	LOCAL CONST Robtarget Tr_meulage_bavure_P251 :=[[98.1400390625,117.987203125,73.8456328125],[0.127040389675562,-0.107005563499621,0.63527191816149,-0.754214915502625],[0,0,0,0],[8.999999E+09,8.999999E+09,8.999999E+09,8.999999E+09,8.999999E+09,8.999999E+09]];
	LOCAL CONST Robtarget Tr_meulage_bavure_P252 :=[[98.0491484375,117.9515,73.860046875],[0.172195881687435,-0.145894069896958,0.629753687846079,-0.74328580730635],[0,0,0,0],[8.999999E+09,8.999999E+09,8.999999E+09,8.999999E+09,8.999999E+09,8.999999E+09]];
	LOCAL CONST Robtarget Tr_meulage_bavure_P253 :=[[95.44875,117.0130703125,74.2617890625],[0.207950204557917,-0.177032849806687,0.623590925198428,-0.73249603447651],[0,0,0,0],[8.999999E+09,8.999999E+09,8.999999E+09,8.999999E+09,8.999999E+09,8.999999E+09]];
	LOCAL CONST Robtarget Tr_meulage_bavure_P254 :=[[94.7231171875,116.4957578125,74.4063515625],[0.235260133644742,-0.200979067526871,0.617662145956152,-0.72301698277864],[0,0,0,0],[8.999999E+09,8.999999E+09,8.999999E+09,8.999999E+09,8.999999E+09,8.999999E+09]];
	LOCAL CONST Robtarget Tr_meulage_bavure_P255 :=[[94.14340625,116.1705234375,74.51065625],[0.255147496976429,-0.218409662757732,0.612521728241192,-0.715551609901858],[0,0,0,0],[8.999999E+09,8.999999E+09,8.999999E+09,8.999999E+09,8.999999E+09,8.999999E+09]];
	LOCAL CONST Robtarget Tr_meulage_bavure_P256 :=[[93.2889140625,115.3411484375,74.708875],[0.268575710211451,-0.230015700629152,0.608452712166897,-0.710454194445527],[0,0,0,0],[8.999999E+09,8.999999E+09,8.999999E+09,8.999999E+09,8.999999E+09,8.999999E+09]];
	LOCAL CONST Robtarget Tr_meulage_bavure_P257 :=[[90.7856171875,112.887015625,75.292671875],[0.276376961310427,-0.236441862806716,0.605550122499022,-0.707827712025126],[0,0,0,0],[8.999999E+09,8.999999E+09,8.999999E+09,8.999999E+09,8.999999E+09,8.999999E+09]];
	LOCAL CONST Robtarget Tr_meulage_bavure_P258 :=[[88.863078125,110.5822109375,75.79440625],[0.279245959102819,-0.238275525006702,0.603780767368518,-0.707598228844173],[0,0,0,0],[8.999999E+09,8.999999E+09,8.999999E+09,8.999999E+09,8.999999E+09,8.999999E+09]];
	LOCAL CONST Robtarget Tr_meulage_bavure_P259 :=[[86.18025,107.824984375,76.4362265625],[0.277632487950623,-0.235945820214436,0.603068641778131,-0.709618196540621],[0,0,0,0],[8.999999E+09,8.999999E+09,8.999999E+09,8.999999E+09,8.999999E+09,8.999999E+09]];
	LOCAL CONST Robtarget Tr_meulage_bavure_P260 :=[[80.36984375,101.8534296875,77.8262578125],[0.27163574756326,-0.229638288909727,0.603381148543333,-0.713730668035842],[0,0,0,0],[8.999999E+09,8.999999E+09,8.999999E+09,8.999999E+09,8.999999E+09,8.999999E+09]];
	LOCAL CONST Robtarget Tr_meulage_bavure_P261 :=[[77.1337109375,98.5814375,78.59359375],[0.260925476383616,-0.219208728105446,0.60474203438692,-0.719828105273714],[0,0,0,0],[8.999999E+09,8.999999E+09,8.999999E+09,8.999999E+09,8.999999E+09,8.999999E+09]];
	LOCAL CONST Robtarget Tr_meulage_bavure_P262 :=[[72.1760859375,93.4272109375,79.787125],[0.244696261183989,-0.204145790459714,0.607216023498567,-0.727830293960579],[0,0,0,0],[8.999999E+09,8.999999E+09,8.999999E+09,8.999999E+09,8.999999E+09,8.999999E+09]];
	LOCAL CONST Robtarget Tr_meulage_bavure_P263 :=[[71.50584375,92.7481328125,79.946234375],[0.221726143472033,-0.183626372472933,0.610829559169254,-0.737567706911403],[0,0,0,0],[8.999999E+09,8.999999E+09,8.999999E+09,8.999999E+09,8.999999E+09,8.999999E+09]];
	LOCAL CONST Robtarget Tr_meulage_bavure_P264 :=[[71.2399140625,92.5131875,80.0049765625],[0.190628848170377,-0.156707517312216,0.615389383499725,-0.748598225311084],[0,0,0,0],[8.999999E+09,8.999999E+09,8.999999E+09,8.999999E+09,8.999999E+09,8.999999E+09]];
	LOCAL CONST Robtarget Tr_meulage_bavure_P265 :=[[70.7853359375,92.1913046875,80.0952578125],[0.150575822021713,-0.122909725316936,0.620287722757024,-0.759910035623892],[0,0,0,0],[8.999999E+09,8.999999E+09,8.999999E+09,8.999999E+09,8.999999E+09,8.999999E+09]];
	LOCAL CONST Robtarget Tr_meulage_bavure_P266 :=[[68.07696875,90.16765625,80.6466328125],[0.102447611715575,-0.0830907118710058,0.624412481473696,-0.769876271510173],[0,0,0,0],[8.999999E+09,8.999999E+09,8.999999E+09,8.999999E+09,8.999999E+09,8.999999E+09]];
	LOCAL CONST Robtarget Tr_meulage_bavure_P267 :=[[65.683109375,88.9370859375,81.0630625],[0.0497692839972195,-0.0401467777631947,0.626564781602221,-0.776741803343555],[0,0,0,0],[8.999999E+09,8.999999E+09,8.999999E+09,8.999999E+09,8.999999E+09,8.999999E+09]];
	LOCAL CONST Robtarget Tr_meulage_bavure_P268 :=[[64.74205859375,88.55846875,81.21340625],[0.001363095089986,-0.00109499953132052,-0.626270337472808,0.779604006755672],[0,0,0,0],[8.999999E+09,8.999999E+09,8.999999E+09,8.999999E+09,8.999999E+09,8.999999E+09]];
	LOCAL CONST Robtarget Tr_meulage_bavure_P269 :=[[62.3850234375,88.1528203125,81.5210078125],[0.0437419301601574,-0.0350453753396799,-0.624275842926536,0.779190693701823],[0,0,0,0],[8.999999E+09,8.999999E+09,8.999999E+09,8.999999E+09,8.999999E+09,8.999999E+09]];
	LOCAL CONST Robtarget Tr_meulage_bavure_P270 :=[[61.54280859375,88.344234375,81.5881796875],[0.0710459531376083,-0.0568640478748205,-0.622285158362753,0.777483205145618],[0,0,0,0],[8.999999E+09,8.999999E+09,8.999999E+09,8.999999E+09,8.999999E+09,8.999999E+09]];
	LOCAL CONST Robtarget Tr_meulage_bavure_P271 :=[[59.371765625,88.1027109375,81.85471875],[0.0786620779021897,-0.0630080775834088,-0.621986088766345,0.776515012759249],[0,0,0,0],[8.999999E+09,8.999999E+09,8.999999E+09,8.999999E+09,8.999999E+09,8.999999E+09]];
	LOCAL CONST Robtarget Tr_meulage_bavure_P272 :=[[56.79593359375,90.4163515625,81.840546875],[0.064068817064071,-0.0514508699376922,-0.624029588381331,0.777068251498729],[0,0,0,0],[8.999999E+09,8.999999E+09,8.999999E+09,8.999999E+09,8.999999E+09,8.999999E+09]];
	LOCAL CONST Robtarget Tr_meulage_bavure_P273 :=[[48.6920625,97.4299765625,81.8296640625],[0.0277015568674016,-0.0223423861530457,-0.62739597405027,0.777886709793671],[0,0,0,0],[8.999999E+09,8.999999E+09,8.999999E+09,8.999999E+09,8.999999E+09,8.999999E+09]];
	LOCAL CONST Robtarget Tr_meulage_bavure_P274 :=[[47.0812421875,97.794265625,81.9583671875],[0.0252356318326453,-0.0204756378074699,0.629734896885263,-0.776130060484254],[0,0,0,0],[8.999999E+09,8.999999E+09,8.999999E+09,8.999999E+09,8.999999E+09,8.999999E+09]];
	LOCAL CONST Robtarget Tr_meulage_bavure_P275 :=[[44.806,97.7003515625,82.21746875],[0.0848193325394842,-0.0693367803526094,0.629095491043596,-0.769569330773068],[0,0,0,0],[8.999999E+09,8.999999E+09,8.999999E+09,8.999999E+09,8.999999E+09,8.999999E+09]];
	LOCAL CONST Robtarget Tr_meulage_bavure_P276 :=[[42.50455859375,97.2184921875,82.52871875],[0.140587062127015,-0.115938530664608,0.625580695787566,-0.758579150865466],[0,0,0,0],[8.999999E+09,8.999999E+09,8.999999E+09,8.999999E+09,8.999999E+09,8.999999E+09]];
	LOCAL CONST Robtarget Tr_meulage_bavure_P277 :=[[39.54287109375,95.636578125,83.0514765625],[0.186282650440504,-0.155136411224339,0.620854079163028,-0.745500959384978],[0,0,0,0],[8.999999E+09,8.999999E+09,8.999999E+09,8.999999E+09,8.999999E+09,8.999999E+09]];
	LOCAL CONST Robtarget Tr_meulage_bavure_P278 :=[[39.0804296875,95.4284609375,83.1281640625],[0.220511472840555,-0.185597052614264,0.616612847403539,-0.732609732957109],[0,0,0,0],[8.999999E+09,8.999999E+09,8.999999E+09,8.999999E+09,8.999999E+09,8.999999E+09]];
	LOCAL CONST Robtarget Tr_meulage_bavure_P279 :=[[38.82609765625,95.2573359375,83.1775390625],[0.244591306708348,-0.208162312657775,0.613779305281082,-0.721192421396913],[0,0,0,0],[8.999999E+09,8.999999E+09,8.999999E+09,8.999999E+09,8.999999E+09,8.999999E+09]];
	LOCAL CONST Robtarget Tr_meulage_bavure_P280 :=[[35.845515625,92.55171875,83.845140625],[0.260660984276943,-0.224358974738056,0.612563122723334,-0.711677822058339],[0,0,0,0],[8.999999E+09,8.999999E+09,8.999999E+09,8.999999E+09,8.999999E+09,8.999999E+09]];
	LOCAL CONST Robtarget Tr_meulage_bavure_P281 :=[[32.57470703125,88.9592421875,84.65696875],[0.270796308543816,-0.235720468748974,0.61279461348127,-0.703980100272833],[0,0,0,0],[8.999999E+09,8.999999E+09,8.999999E+09,8.999999E+09,8.999999E+09,8.999999E+09]];
	LOCAL CONST Robtarget Tr_meulage_bavure_P282 :=[[32.4998046875,88.8786796875,84.67534375],[0.276769983598911,-0.243580619288763,0.614120686336212,-0.697798424116522],[0,0,0,0],[8.999999E+09,8.999999E+09,8.999999E+09,8.999999E+09,8.999999E+09,8.999999E+09]];
	LOCAL CONST Robtarget Tr_meulage_bavure_P283 :=[[32.41517578125,88.7886328125,84.6959765625],[0.279976048156399,-0.249000355415884,0.616150254112905,-0.692799465803844],[0,0,0,0],[8.999999E+09,8.999999E+09,8.999999E+09,8.999999E+09,8.999999E+09,8.999999E+09]];
	LOCAL CONST Robtarget Tr_meulage_bavure_P284 :=[[32.27737890625,88.6504765625,84.7285078125],[0.281492307641199,-0.252818582194378,0.618524049054791,-0.688674702582376],[0,0,0,0],[8.999999E+09,8.999999E+09,8.999999E+09,8.999999E+09,8.999999E+09,8.999999E+09]];
	LOCAL CONST Robtarget Tr_meulage_bavure_P285 :=[[28.927525390625,85.261125,85.523109375],[0.282090145605153,-0.255653636684952,0.620965252888204,-0.685177730598208],[0,0,0,0],[8.999999E+09,8.999999E+09,8.999999E+09,8.999999E+09,8.999999E+09,8.999999E+09]];
	LOCAL CONST Robtarget Tr_meulage_bavure_P286 :=[[21.47466796875,77.75175,87.286984375],[0.282327813795655,-0.257956584167709,0.623251031261927,-0.682134560239282],[0,0,0,0],[8.999999E+09,8.999999E+09,8.999999E+09,8.999999E+09,8.999999E+09,8.999999E+09]];
	LOCAL CONST Robtarget Tr_meulage_bavure_P287 :=[[21.25967578125,77.5322421875,87.338234375],[0.282601819625309,-0.260063837576601,0.625225023955301,-0.679409067756303],[0,0,0,0],[8.999999E+09,8.999999E+09,8.999999E+09,8.999999E+09,8.999999E+09,8.999999E+09]];
	LOCAL CONST Robtarget Tr_meulage_bavure_P288 :=[[20.5857109375,76.868484375,87.495796875],[0.283101282414858,-0.26214225566945,0.626816081849102,-0.67693182908099],[0,0,0,0],[8.999999E+09,8.999999E+09,8.999999E+09,8.999999E+09,8.999999E+09,8.999999E+09]];
	LOCAL CONST Robtarget Tr_meulage_bavure_P289 :=[[16.90142578125,73.2369765625,88.3575],[0.283868643218972,-0.264223838178046,0.628004469387492,-0.674696037608653],[0,0,0,0],[8.999999E+09,8.999999E+09,8.999999E+09,8.999999E+09,8.999999E+09,8.999999E+09]];
	LOCAL CONST Robtarget Tr_meulage_bavure_P290 :=[[15.873087890625,72.23375,88.5966953125],[0.284822251592282,-0.26622897396762,0.628823532756499,-0.672740204737079],[0,0,0,0],[8.999999E+09,8.999999E+09,8.999999E+09,8.999999E+09,8.999999E+09,8.999999E+09]];
	LOCAL CONST Robtarget Tr_meulage_bavure_P291 :=[[15.2935966796875,71.60771875,88.739203125],[0.285799359935917,-0.268004907206124,0.629345060745857,-0.671131052841732],[0,0,0,0],[8.999999E+09,8.999999E+09,8.999999E+09,8.999999E+09,8.999999E+09,8.999999E+09]];
	LOCAL CONST Robtarget Tr_meulage_bavure_P292 :=[[12.464833984375,68.6040234375,89.4281953125],[0.286627272536143,-0.269395860937951,0.629654783981739,-0.669929496109032],[0,0,0,0],[8.999999E+09,8.999999E+09,8.999999E+09,8.999999E+09,8.999999E+09,8.999999E+09]];
	LOCAL CONST Robtarget Tr_meulage_bavure_P293 :=[[12.3877333984375,68.5313046875,89.4458046875],[0.287172673957076,-0.270282218475825,0.629822260816589,-0.669181064800857],[0,0,0,0],[8.999999E+09,8.999999E+09,8.999999E+09,8.999999E+09,8.999999E+09,8.999999E+09]];
	LOCAL CONST Robtarget Tr_meulage_bavure_P294 :=[[12.30885546875,68.4598515625,89.463453125],[0.287361487578792,-0.270586373771854,0.629876519961336,-0.668925974519527],[0,0,0,0],[8.999999E+09,8.999999E+09,8.999999E+09,8.999999E+09,8.999999E+09,8.999999E+09]];
	LOCAL CONST Robtarget Tr_meulage_bavure_degg1 :=[[5.0687653180683,75.3315448036295,88.8626814463921],[0.287361487578792,-0.270586373771854,0.629876519961336,-0.668925974519527],[0,0,0,0],[8.999999E+09,8.999999E+09,8.999999E+09,8.999999E+09,8.999999E+09,8.999999E+09]];
	LOCAL CONST Robtarget Tr_meulage_bavure_degg2 :=[[-132.492947544884,205.89371638509,77.4480195528422],[0.287361487578792,-0.270586373771854,0.629876519961336,-0.668925974519527],[0,0,0,0],[8.999999E+09,8.999999E+09,8.999999E+09,8.999999E+09,8.999999E+09,8.999999E+09]];
	LOCAL PROC Tr_pick()
		!!Programme Tr_pick - 11/05/2023 15:21:44;
		 CONST Robtarget Ppick :=[[54.302843354765,-14.0729442667339,117.853362865586],[0.0438323717266724,0.92362905790366,0.371077115821677,-0.0853806810600477],[0,0,0,0],[8.999999E+09,8.999999E+09,8.999999E+09,8.999999E+09,8.999999E+09,8.999999E+09]];
		 VAR Pose Ref :=[[0,0,0],[1,0,0,0]];
		LocalisationPieceTable 80 \model:=0;
		MoveJ Reltool(Ppick,0,0,-200),V1000,Z0,Tool_Prehenseur_1 \Wobj:=Wobj_vision;
		MoveL Reltool(Ppick,0,0,-100),V500,Z0,Tool_Prehenseur_1 \Wobj:=Wobj_vision;
		MoveL Reltool(Ppick,0,0,-10),V200,Z0,Tool_Prehenseur_1 \Wobj:=Wobj_vision;
		MoveL Ppick,V100,Fine,Tool_Prehenseur_1 \Wobj:=Wobj_vision;
		Gripper_Close;
		MoveL Reltool(Ppick,0,0,-200),V500,Z0,Tool_Prehenseur_1 \Wobj:=Wobj_vision;
		LocalisationPiecePrehenseur 80 \model:=0,Ref;
	ENDPROC
	LOCAL PROC Tr_Cut()
		!!Programme Tr_Cut - 11/05/2023 15:21:44;
		confJ \off;
		confL \off;
		Tool := ToolOffset(Tool_M2_D490_S180);
	ENDPROC
	LOCAL PROC Tr_meulage_motif_1()
		!!Programme Tr_meulage_motif_1 - 11/05/2023 15:21:44;
		 CONST Speeddata vitesse_Meulage :=[50, 500, 0, 0];
		confJ \off;
		confL \off;
		Tool := ToolOffset(Tool_M1_D500_S0);
		MoveAbsJ [[0,-40,40,0,90,0],[8.999999E+09,8.999999E+09,8.999999E+09,8.999999E+09,8.999999E+09,8.999999E+09]] ,V1000,Z0,Tool_M1_D500_S0 \Wobj:=Wobj_Part_0;
		MoveJ Tr_meulage_motif_1_App1,V2000,Z100,Tool,\Wobj:=Wobj_Part_0;
		MoveJ Tr_meulage_motif_1_App2,V500,Z0,Tool,\Wobj:=Wobj_Part_0;
		MoveL Tr_meulage_motif_1_P0,[12.5,500,0,0],z0,Tool \wobj:=Wobj_Part_0;
		MoveL Tr_meulage_motif_1_P1,[12.5,500,0,0],z0,Tool \wobj:=Wobj_Part_0;
		MoveL Tr_meulage_motif_1_P2,[12.5,500,0,0],z0,Tool \wobj:=Wobj_Part_0;
		MoveL Tr_meulage_motif_1_P3,[12.5,500,0,0],z0,Tool \wobj:=Wobj_Part_0;
		MoveL Tr_meulage_motif_1_P4,[12.5,500,0,0],z0,Tool \wobj:=Wobj_Part_0;
		MoveL Tr_meulage_motif_1_P5,[12.5,500,0,0],z0,Tool \wobj:=Wobj_Part_0;
		MoveL Tr_meulage_motif_1_P6,[12.5,500,0,0],z0,Tool \wobj:=Wobj_Part_0;
		MoveL Tr_meulage_motif_1_P7,[12.5,500,0,0],z0,Tool \wobj:=Wobj_Part_0;
		MoveL Tr_meulage_motif_1_P8,[12.5,500,0,0],z0,Tool \wobj:=Wobj_Part_0;
		MoveL Tr_meulage_motif_1_P9,[12.5,500,0,0],z0,Tool \wobj:=Wobj_Part_0;
		MoveL Tr_meulage_motif_1_P10,[12.5,500,0,0],z0,Tool \wobj:=Wobj_Part_0;
		MoveL Tr_meulage_motif_1_P11,[12.5,500,0,0],z0,Tool \wobj:=Wobj_Part_0;
		MoveL Tr_meulage_motif_1_P12,[12.5,500,0,0],z0,Tool \wobj:=Wobj_Part_0;
		MoveL Tr_meulage_motif_1_P13,[12.5,500,0,0],z0,Tool \wobj:=Wobj_Part_0;
		MoveL Tr_meulage_motif_1_P14,[12.5,500,0,0],z0,Tool \wobj:=Wobj_Part_0;
		MoveL Tr_meulage_motif_1_P15,[12.5,500,0,0],z0,Tool \wobj:=Wobj_Part_0;
		MoveL Tr_meulage_motif_1_P16,[12.5,500,0,0],z0,Tool \wobj:=Wobj_Part_0;
		MoveL Tr_meulage_motif_1_P17,[12.5,500,0,0],z0,Tool \wobj:=Wobj_Part_0;
		MoveL Tr_meulage_motif_1_P18,[12.5,500,0,0],z0,Tool \wobj:=Wobj_Part_0;
		MoveL Tr_meulage_motif_1_P19,[12.5,500,0,0],z0,Tool \wobj:=Wobj_Part_0;
		MoveL Tr_meulage_motif_1_P20,[12.5,500,0,0],z0,Tool \wobj:=Wobj_Part_0;
		MoveL Tr_meulage_motif_1_P21,[12.5,500,0,0],z0,Tool \wobj:=Wobj_Part_0;
		MoveL Tr_meulage_motif_1_P22,[12.5,500,0,0],z0,Tool \wobj:=Wobj_Part_0;
		MoveL Tr_meulage_motif_1_P23,[12.5,500,0,0],z0,Tool \wobj:=Wobj_Part_0;
		MoveL Tr_meulage_motif_1_P24,[12.5,500,0,0],z0,Tool \wobj:=Wobj_Part_0;
		MoveL Tr_meulage_motif_1_P25,[12.5,500,0,0],z0,Tool \wobj:=Wobj_Part_0;
		MoveL Tr_meulage_motif_1_P26,[12.5,500,0,0],z0,Tool \wobj:=Wobj_Part_0;
		MoveL Tr_meulage_motif_1_P27,[12.5,500,0,0],z0,Tool \wobj:=Wobj_Part_0;
		MoveL Tr_meulage_motif_1_P28,[12.5,500,0,0],z0,Tool \wobj:=Wobj_Part_0;
		MoveL Tr_meulage_motif_1_P29,[12.5,500,0,0],z0,Tool \wobj:=Wobj_Part_0;
		MoveL Tr_meulage_motif_1_P30,[12.5,500,0,0],z0,Tool \wobj:=Wobj_Part_0;
		MoveL Tr_meulage_motif_1_P31,[12.5,500,0,0],z0,Tool \wobj:=Wobj_Part_0;
		MoveL Tr_meulage_motif_1_P32,[12.5,500,0,0],z0,Tool \wobj:=Wobj_Part_0;
		MoveL Tr_meulage_motif_1_P33,[12.5,500,0,0],z0,Tool \wobj:=Wobj_Part_0;
		MoveL Tr_meulage_motif_1_P34,[12.5,500,0,0],z0,Tool \wobj:=Wobj_Part_0;
		MoveL Tr_meulage_motif_1_P35,[12.5,500,0,0],z0,Tool \wobj:=Wobj_Part_0;
		MoveL Tr_meulage_motif_1_P36,[12.5,500,0,0],z0,Tool \wobj:=Wobj_Part_0;
		MoveL Tr_meulage_motif_1_P37,[12.5,500,0,0],z0,Tool \wobj:=Wobj_Part_0;
		MoveL Tr_meulage_motif_1_P38,[12.5,500,0,0],z0,Tool \wobj:=Wobj_Part_0;
		MoveL Tr_meulage_motif_1_P39,[12.5,500,0,0],z0,Tool \wobj:=Wobj_Part_0;
		MoveL Tr_meulage_motif_1_P40,[12.5,500,0,0],z0,Tool \wobj:=Wobj_Part_0;
		MoveL Tr_meulage_motif_1_P41,[12.5,500,0,0],z0,Tool \wobj:=Wobj_Part_0;
		MoveL Tr_meulage_motif_1_P42,[12.5,500,0,0],z0,Tool \wobj:=Wobj_Part_0;
		MoveL Tr_meulage_motif_1_P43,[12.5,500,0,0],z0,Tool \wobj:=Wobj_Part_0;
		MoveL Tr_meulage_motif_1_P44,[12.5,500,0,0],z0,Tool \wobj:=Wobj_Part_0;
		MoveL Tr_meulage_motif_1_P45,[12.5,500,0,0],z0,Tool \wobj:=Wobj_Part_0;
		MoveL Tr_meulage_motif_1_P46,[12.5,500,0,0],z0,Tool \wobj:=Wobj_Part_0;
		MoveL Tr_meulage_motif_1_P47,[12.5,500,0,0],z0,Tool \wobj:=Wobj_Part_0;
		MoveL Tr_meulage_motif_1_P48,[12.5,500,0,0],z0,Tool \wobj:=Wobj_Part_0;
		MoveL Tr_meulage_motif_1_P49,[12.5,500,0,0],z0,Tool \wobj:=Wobj_Part_0;
		MoveL Tr_meulage_motif_1_P50,[12.5,500,0,0],z0,Tool \wobj:=Wobj_Part_0;
		MoveL Tr_meulage_motif_1_P51,[12.5,500,0,0],z0,Tool \wobj:=Wobj_Part_0;
		MoveL Tr_meulage_motif_1_P52,[12.5,500,0,0],z0,Tool \wobj:=Wobj_Part_0;
		MoveL Tr_meulage_motif_1_P53,[12.5,500,0,0],z0,Tool \wobj:=Wobj_Part_0;
		MoveL Tr_meulage_motif_1_P54,[12.5,500,0,0],z0,Tool \wobj:=Wobj_Part_0;
		MoveL Tr_meulage_motif_1_P55,[12.5,500,0,0],z0,Tool \wobj:=Wobj_Part_0;
		MoveL Tr_meulage_motif_1_P56,[12.5,500,0,0],z0,Tool \wobj:=Wobj_Part_0;
		MoveL Tr_meulage_motif_1_P57,[12.5,500,0,0],z0,Tool \wobj:=Wobj_Part_0;
		MoveL Tr_meulage_motif_1_P58,[12.5,500,0,0],z0,Tool \wobj:=Wobj_Part_0;
		MoveL Tr_meulage_motif_1_P59,[12.5,500,0,0],z0,Tool \wobj:=Wobj_Part_0;
		MoveL Tr_meulage_motif_1_P60,[12.5,500,0,0],z0,Tool \wobj:=Wobj_Part_0;
		MoveL Tr_meulage_motif_1_P61,[12.5,500,0,0],z0,Tool \wobj:=Wobj_Part_0;
		MoveL Tr_meulage_motif_1_P62,[12.5,500,0,0],z0,Tool \wobj:=Wobj_Part_0;
		MoveL Tr_meulage_motif_1_P63,[12.5,500,0,0],z0,Tool \wobj:=Wobj_Part_0;
		MoveL Tr_meulage_motif_1_P64,[12.5,500,0,0],z0,Tool \wobj:=Wobj_Part_0;
		MoveL Tr_meulage_motif_1_P65,[12.5,500,0,0],z0,Tool \wobj:=Wobj_Part_0;
		MoveL Tr_meulage_motif_1_P66,[12.5,500,0,0],z0,Tool \wobj:=Wobj_Part_0;
		MoveL Tr_meulage_motif_1_P67,[12.5,500,0,0],z0,Tool \wobj:=Wobj_Part_0;
		MoveL Tr_meulage_motif_1_P68,[12.5,500,0,0],z0,Tool \wobj:=Wobj_Part_0;
		MoveL Tr_meulage_motif_1_P69,[12.5,500,0,0],z0,Tool \wobj:=Wobj_Part_0;
		MoveL Tr_meulage_motif_1_P70,[12.5,500,0,0],z0,Tool \wobj:=Wobj_Part_0;
		MoveL Tr_meulage_motif_1_P71,[12.5,500,0,0],z0,Tool \wobj:=Wobj_Part_0;
		MoveL Tr_meulage_motif_1_P72,[12.5,500,0,0],z0,Tool \wobj:=Wobj_Part_0;
		MoveL Tr_meulage_motif_1_P73,[12.5,500,0,0],z0,Tool \wobj:=Wobj_Part_0;
		MoveL Tr_meulage_motif_1_P74,[12.5,500,0,0],z0,Tool \wobj:=Wobj_Part_0;
		MoveL Tr_meulage_motif_1_P75,[12.5,500,0,0],z0,Tool \wobj:=Wobj_Part_0;
		MoveL Tr_meulage_motif_1_P76,[12.5,500,0,0],z0,Tool \wobj:=Wobj_Part_0;
		MoveL Tr_meulage_motif_1_P77,[12.5,500,0,0],z0,Tool \wobj:=Wobj_Part_0;
		MoveL Tr_meulage_motif_1_P78,[12.5,500,0,0],z0,Tool \wobj:=Wobj_Part_0;
		MoveL Tr_meulage_motif_1_P79,[12.5,500,0,0],z0,Tool \wobj:=Wobj_Part_0;
		MoveL Tr_meulage_motif_1_P80,[12.5,500,0,0],z0,Tool \wobj:=Wobj_Part_0;
		MoveL Tr_meulage_motif_1_P81,[12.5,500,0,0],z0,Tool \wobj:=Wobj_Part_0;
		MoveL Tr_meulage_motif_1_P82,[12.5,500,0,0],z0,Tool \wobj:=Wobj_Part_0;
		MoveL Tr_meulage_motif_1_P83,[12.5,500,0,0],z0,Tool \wobj:=Wobj_Part_0;
		MoveL Tr_meulage_motif_1_P84,[12.5,500,0,0],z0,Tool \wobj:=Wobj_Part_0;
		MoveL Tr_meulage_motif_1_P85,[12.5,500,0,0],z0,Tool \wobj:=Wobj_Part_0;
		MoveL Tr_meulage_motif_1_P86,[12.5,500,0,0],z0,Tool \wobj:=Wobj_Part_0;
		MoveL Tr_meulage_motif_1_P87,[12.5,500,0,0],z0,Tool \wobj:=Wobj_Part_0;
		MoveL Tr_meulage_motif_1_P88,[12.5,500,0,0],z0,Tool \wobj:=Wobj_Part_0;
		MoveL Tr_meulage_motif_1_P89,[12.5,500,0,0],z0,Tool \wobj:=Wobj_Part_0;
		MoveL Tr_meulage_motif_1_P90,[12.5,500,0,0],z0,Tool \wobj:=Wobj_Part_0;
		MoveL Tr_meulage_motif_1_P91,[12.5,500,0,0],z0,Tool \wobj:=Wobj_Part_0;
		MoveL Tr_meulage_motif_1_P92,[12.5,500,0,0],z0,Tool \wobj:=Wobj_Part_0;
		MoveL Tr_meulage_motif_1_P93,[12.5,500,0,0],z0,Tool \wobj:=Wobj_Part_0;
		MoveL Tr_meulage_motif_1_P94,[12.5,500,0,0],z0,Tool \wobj:=Wobj_Part_0;
		MoveL Tr_meulage_motif_1_P95,[12.5,500,0,0],z0,Tool \wobj:=Wobj_Part_0;
		MoveL Tr_meulage_motif_1_P96,[12.5,500,0,0],z0,Tool \wobj:=Wobj_Part_0;
		MoveL Tr_meulage_motif_1_P97,[12.5,500,0,0],z0,Tool \wobj:=Wobj_Part_0;
		MoveL Tr_meulage_motif_1_P98,[12.5,500,0,0],z0,Tool \wobj:=Wobj_Part_0;
		MoveL Tr_meulage_motif_1_P99,[12.5,500,0,0],z0,Tool \wobj:=Wobj_Part_0;
		MoveL Tr_meulage_motif_1_P100,[12.5,500,0,0],z0,Tool \wobj:=Wobj_Part_0;
		MoveL Tr_meulage_motif_1_P101,[12.5,500,0,0],z0,Tool \wobj:=Wobj_Part_0;
		MoveL Tr_meulage_motif_1_P102,[12.5,500,0,0],z0,Tool \wobj:=Wobj_Part_0;
		MoveL Tr_meulage_motif_1_P103,[12.5,500,0,0],z0,Tool \wobj:=Wobj_Part_0;
		MoveL Tr_meulage_motif_1_P104,[12.5,500,0,0],z0,Tool \wobj:=Wobj_Part_0;
		MoveL Tr_meulage_motif_1_P105,[12.5,500,0,0],z0,Tool \wobj:=Wobj_Part_0;
		MoveL Tr_meulage_motif_1_P106,[12.5,500,0,0],z0,Tool \wobj:=Wobj_Part_0;
		MoveL Tr_meulage_motif_1_P107,[12.5,500,0,0],z0,Tool \wobj:=Wobj_Part_0;
		MoveL Tr_meulage_motif_1_P108,[12.5,500,0,0],z0,Tool \wobj:=Wobj_Part_0;
		MoveL Tr_meulage_motif_1_P109,[12.5,500,0,0],z0,Tool \wobj:=Wobj_Part_0;
		MoveL Tr_meulage_motif_1_P110,[12.5,500,0,0],z0,Tool \wobj:=Wobj_Part_0;
		MoveL Tr_meulage_motif_1_P111,[12.5,500,0,0],z0,Tool \wobj:=Wobj_Part_0;
		MoveL Tr_meulage_motif_1_P112,[12.5,500,0,0],z0,Tool \wobj:=Wobj_Part_0;
		MoveL Tr_meulage_motif_1_P113,[12.5,500,0,0],z0,Tool \wobj:=Wobj_Part_0;
		MoveL Tr_meulage_motif_1_P114,[12.5,500,0,0],z0,Tool \wobj:=Wobj_Part_0;
		MoveL Tr_meulage_motif_1_P115,[12.5,500,0,0],z0,Tool \wobj:=Wobj_Part_0;
		MoveL Tr_meulage_motif_1_P116,[12.5,500,0,0],z0,Tool \wobj:=Wobj_Part_0;
		MoveL Tr_meulage_motif_1_P117,[12.5,500,0,0],z0,Tool \wobj:=Wobj_Part_0;
		MoveL Tr_meulage_motif_1_P118,[12.5,500,0,0],z0,Tool \wobj:=Wobj_Part_0;
		MoveL Tr_meulage_motif_1_P119,[12.5,500,0,0],z0,Tool \wobj:=Wobj_Part_0;
		MoveL Tr_meulage_motif_1_P120,[12.5,500,0,0],z0,Tool \wobj:=Wobj_Part_0;
		MoveL Tr_meulage_motif_1_P121,[12.5,500,0,0],z0,Tool \wobj:=Wobj_Part_0;
		MoveL Tr_meulage_motif_1_P122,[12.5,500,0,0],z0,Tool \wobj:=Wobj_Part_0;
		MoveL Tr_meulage_motif_1_P123,[12.5,500,0,0],z0,Tool \wobj:=Wobj_Part_0;
		MoveJ Tr_meulage_motif_1_degg1,V500,Z0,Tool,\Wobj:=Wobj_Part_0;
		MoveJ Tr_meulage_motif_1_degg2,V2000,Z100,Tool,\Wobj:=Wobj_Part_0;
	ENDPROC
	LOCAL PROC Tr_meulage_bavure()
		!!Programme Tr_meulage_bavure - 11/05/2023 15:21:44;
		 CONST Speeddata vitesse_Meulage :=[50, 500, 0, 0];
		confJ \off;
		confL \off;
		Tool := ToolOffset(Tool_M1_D500_S0);
		MoveAbsJ [[0,-40,40,0,90,0],[8.999999E+09,8.999999E+09,8.999999E+09,8.999999E+09,8.999999E+09,8.999999E+09]] ,V1000,Z0,Tool_M1_D500_S0 \Wobj:=Wobj_Part_0;
		MoveJ Tr_meulage_bavure_App1,V2000,Z100,Tool,\Wobj:=Wobj_Part_0;
		MoveJ Tr_meulage_bavure_App2,V500,Z0,Tool,\Wobj:=Wobj_Part_0;
		MoveL Tr_meulage_bavure_P0,[50,500,0,0],z0,Tool \wobj:=Wobj_Part_0;
		MoveL Tr_meulage_bavure_P1,[50,500,0,0],z0,Tool \wobj:=Wobj_Part_0;
		MoveL Tr_meulage_bavure_P2,[50,500,0,0],z0,Tool \wobj:=Wobj_Part_0;
		MoveL Tr_meulage_bavure_P3,[50,500,0,0],z0,Tool \wobj:=Wobj_Part_0;
		MoveL Tr_meulage_bavure_P4,[50,500,0,0],z0,Tool \wobj:=Wobj_Part_0;
		MoveL Tr_meulage_bavure_P5,[50,500,0,0],z0,Tool \wobj:=Wobj_Part_0;
		MoveL Tr_meulage_bavure_P6,[50,500,0,0],z0,Tool \wobj:=Wobj_Part_0;
		MoveL Tr_meulage_bavure_P7,[50,500,0,0],z0,Tool \wobj:=Wobj_Part_0;
		MoveL Tr_meulage_bavure_P8,[50,500,0,0],z0,Tool \wobj:=Wobj_Part_0;
		MoveL Tr_meulage_bavure_P9,[50,500,0,0],z0,Tool \wobj:=Wobj_Part_0;
		MoveL Tr_meulage_bavure_P10,[50,500,0,0],z0,Tool \wobj:=Wobj_Part_0;
		MoveL Tr_meulage_bavure_P11,[50,500,0,0],z0,Tool \wobj:=Wobj_Part_0;
		MoveL Tr_meulage_bavure_P12,[50,500,0,0],z0,Tool \wobj:=Wobj_Part_0;
		MoveL Tr_meulage_bavure_P13,[50,500,0,0],z0,Tool \wobj:=Wobj_Part_0;
		MoveL Tr_meulage_bavure_P14,[50,500,0,0],z0,Tool \wobj:=Wobj_Part_0;
		MoveL Tr_meulage_bavure_P15,[50,500,0,0],z0,Tool \wobj:=Wobj_Part_0;
		MoveL Tr_meulage_bavure_P16,[50,500,0,0],z0,Tool \wobj:=Wobj_Part_0;
		MoveL Tr_meulage_bavure_P17,[50,500,0,0],z0,Tool \wobj:=Wobj_Part_0;
		MoveL Tr_meulage_bavure_P18,[50,500,0,0],z0,Tool \wobj:=Wobj_Part_0;
		MoveL Tr_meulage_bavure_P19,[50,500,0,0],z0,Tool \wobj:=Wobj_Part_0;
		MoveL Tr_meulage_bavure_P20,[50,500,0,0],z0,Tool \wobj:=Wobj_Part_0;
		MoveL Tr_meulage_bavure_P21,[50,500,0,0],z0,Tool \wobj:=Wobj_Part_0;
		MoveL Tr_meulage_bavure_P22,[50,500,0,0],z0,Tool \wobj:=Wobj_Part_0;
		MoveL Tr_meulage_bavure_P23,[50,500,0,0],z0,Tool \wobj:=Wobj_Part_0;
		MoveL Tr_meulage_bavure_P24,[50,500,0,0],z0,Tool \wobj:=Wobj_Part_0;
		MoveL Tr_meulage_bavure_P25,[50,500,0,0],z0,Tool \wobj:=Wobj_Part_0;
		MoveL Tr_meulage_bavure_P26,[50,500,0,0],z0,Tool \wobj:=Wobj_Part_0;
		MoveL Tr_meulage_bavure_P27,[50,500,0,0],z0,Tool \wobj:=Wobj_Part_0;
		MoveL Tr_meulage_bavure_P28,[50,500,0,0],z0,Tool \wobj:=Wobj_Part_0;
		MoveL Tr_meulage_bavure_P29,[50,500,0,0],z0,Tool \wobj:=Wobj_Part_0;
		MoveL Tr_meulage_bavure_P30,[50,500,0,0],z0,Tool \wobj:=Wobj_Part_0;
		MoveL Tr_meulage_bavure_P31,[50,500,0,0],z0,Tool \wobj:=Wobj_Part_0;
		MoveL Tr_meulage_bavure_P32,[50,500,0,0],z0,Tool \wobj:=Wobj_Part_0;
		MoveL Tr_meulage_bavure_P33,[50,500,0,0],z0,Tool \wobj:=Wobj_Part_0;
		MoveL Tr_meulage_bavure_P34,[50,500,0,0],z0,Tool \wobj:=Wobj_Part_0;
		MoveL Tr_meulage_bavure_P35,[50,500,0,0],z0,Tool \wobj:=Wobj_Part_0;
		MoveL Tr_meulage_bavure_P36,[50,500,0,0],z0,Tool \wobj:=Wobj_Part_0;
		MoveL Tr_meulage_bavure_P37,[50,500,0,0],z0,Tool \wobj:=Wobj_Part_0;
		MoveL Tr_meulage_bavure_P38,[50,500,0,0],z0,Tool \wobj:=Wobj_Part_0;
		MoveL Tr_meulage_bavure_P39,[50,500,0,0],z0,Tool \wobj:=Wobj_Part_0;
		MoveL Tr_meulage_bavure_P40,[50,500,0,0],z0,Tool \wobj:=Wobj_Part_0;
		MoveL Tr_meulage_bavure_P41,[50,500,0,0],z0,Tool \wobj:=Wobj_Part_0;
		MoveL Tr_meulage_bavure_P42,[50,500,0,0],z0,Tool \wobj:=Wobj_Part_0;
		MoveL Tr_meulage_bavure_P43,[50,500,0,0],z0,Tool \wobj:=Wobj_Part_0;
		MoveL Tr_meulage_bavure_P44,[50,500,0,0],z0,Tool \wobj:=Wobj_Part_0;
		MoveL Tr_meulage_bavure_P45,[50,500,0,0],z0,Tool \wobj:=Wobj_Part_0;
		MoveL Tr_meulage_bavure_P46,[50,500,0,0],z0,Tool \wobj:=Wobj_Part_0;
		MoveL Tr_meulage_bavure_P47,[50,500,0,0],z0,Tool \wobj:=Wobj_Part_0;
		MoveL Tr_meulage_bavure_P48,[50,500,0,0],z0,Tool \wobj:=Wobj_Part_0;
		MoveL Tr_meulage_bavure_P49,[50,500,0,0],z0,Tool \wobj:=Wobj_Part_0;
		MoveL Tr_meulage_bavure_P50,[50,500,0,0],z0,Tool \wobj:=Wobj_Part_0;
		MoveL Tr_meulage_bavure_P51,[50,500,0,0],z0,Tool \wobj:=Wobj_Part_0;
		MoveL Tr_meulage_bavure_P52,[50,500,0,0],z0,Tool \wobj:=Wobj_Part_0;
		MoveL Tr_meulage_bavure_P53,[50,500,0,0],z0,Tool \wobj:=Wobj_Part_0;
		MoveL Tr_meulage_bavure_P54,[50,500,0,0],z0,Tool \wobj:=Wobj_Part_0;
		MoveL Tr_meulage_bavure_P55,[50,500,0,0],z0,Tool \wobj:=Wobj_Part_0;
		MoveL Tr_meulage_bavure_P56,[50,500,0,0],z0,Tool \wobj:=Wobj_Part_0;
		MoveL Tr_meulage_bavure_P57,[50,500,0,0],z0,Tool \wobj:=Wobj_Part_0;
		MoveL Tr_meulage_bavure_P58,[50,500,0,0],z0,Tool \wobj:=Wobj_Part_0;
		MoveL Tr_meulage_bavure_P59,[50,500,0,0],z0,Tool \wobj:=Wobj_Part_0;
		MoveL Tr_meulage_bavure_P60,[50,500,0,0],z0,Tool \wobj:=Wobj_Part_0;
		MoveL Tr_meulage_bavure_P61,[50,500,0,0],z0,Tool \wobj:=Wobj_Part_0;
		MoveL Tr_meulage_bavure_P62,[50,500,0,0],z0,Tool \wobj:=Wobj_Part_0;
		MoveL Tr_meulage_bavure_P63,[50,500,0,0],z0,Tool \wobj:=Wobj_Part_0;
		MoveL Tr_meulage_bavure_P64,[50,500,0,0],z0,Tool \wobj:=Wobj_Part_0;
		MoveL Tr_meulage_bavure_P65,[50,500,0,0],z0,Tool \wobj:=Wobj_Part_0;
		MoveL Tr_meulage_bavure_P66,[50,500,0,0],z0,Tool \wobj:=Wobj_Part_0;
		MoveL Tr_meulage_bavure_P67,[50,500,0,0],z0,Tool \wobj:=Wobj_Part_0;
		MoveL Tr_meulage_bavure_P68,[50,500,0,0],z0,Tool \wobj:=Wobj_Part_0;
		MoveL Tr_meulage_bavure_P69,[50,500,0,0],z0,Tool \wobj:=Wobj_Part_0;
		MoveL Tr_meulage_bavure_P70,[50,500,0,0],z0,Tool \wobj:=Wobj_Part_0;
		MoveL Tr_meulage_bavure_P71,[50,500,0,0],z0,Tool \wobj:=Wobj_Part_0;
		MoveL Tr_meulage_bavure_P72,[50,500,0,0],z0,Tool \wobj:=Wobj_Part_0;
		MoveL Tr_meulage_bavure_P73,[50,500,0,0],z0,Tool \wobj:=Wobj_Part_0;
		MoveL Tr_meulage_bavure_P74,[50,500,0,0],z0,Tool \wobj:=Wobj_Part_0;
		MoveL Tr_meulage_bavure_P75,[50,500,0,0],z0,Tool \wobj:=Wobj_Part_0;
		MoveL Tr_meulage_bavure_P76,[50,500,0,0],z0,Tool \wobj:=Wobj_Part_0;
		MoveL Tr_meulage_bavure_P77,[50,500,0,0],z0,Tool \wobj:=Wobj_Part_0;
		MoveL Tr_meulage_bavure_P78,[50,500,0,0],z0,Tool \wobj:=Wobj_Part_0;
		MoveL Tr_meulage_bavure_P79,[50,500,0,0],z0,Tool \wobj:=Wobj_Part_0;
		MoveL Tr_meulage_bavure_P80,[50,500,0,0],z0,Tool \wobj:=Wobj_Part_0;
		MoveL Tr_meulage_bavure_P81,[50,500,0,0],z0,Tool \wobj:=Wobj_Part_0;
		MoveL Tr_meulage_bavure_P82,[50,500,0,0],z0,Tool \wobj:=Wobj_Part_0;
		MoveL Tr_meulage_bavure_P83,[50,500,0,0],z0,Tool \wobj:=Wobj_Part_0;
		MoveL Tr_meulage_bavure_P84,[50,500,0,0],z0,Tool \wobj:=Wobj_Part_0;
		MoveL Tr_meulage_bavure_P85,[50,500,0,0],z0,Tool \wobj:=Wobj_Part_0;
		MoveL Tr_meulage_bavure_P86,[50,500,0,0],z0,Tool \wobj:=Wobj_Part_0;
		MoveL Tr_meulage_bavure_P87,[50,500,0,0],z0,Tool \wobj:=Wobj_Part_0;
		MoveL Tr_meulage_bavure_P88,[50,500,0,0],z0,Tool \wobj:=Wobj_Part_0;
		MoveL Tr_meulage_bavure_P89,[50,500,0,0],z0,Tool \wobj:=Wobj_Part_0;
		MoveL Tr_meulage_bavure_P90,[50,500,0,0],z0,Tool \wobj:=Wobj_Part_0;
		MoveL Tr_meulage_bavure_P91,[50,500,0,0],z0,Tool \wobj:=Wobj_Part_0;
		MoveL Tr_meulage_bavure_P92,[50,500,0,0],z0,Tool \wobj:=Wobj_Part_0;
		MoveL Tr_meulage_bavure_P93,[50,500,0,0],z0,Tool \wobj:=Wobj_Part_0;
		MoveL Tr_meulage_bavure_P94,[50,500,0,0],z0,Tool \wobj:=Wobj_Part_0;
		MoveL Tr_meulage_bavure_P95,[50,500,0,0],z0,Tool \wobj:=Wobj_Part_0;
		MoveL Tr_meulage_bavure_P96,[50,500,0,0],z0,Tool \wobj:=Wobj_Part_0;
		MoveL Tr_meulage_bavure_P97,[50,500,0,0],z0,Tool \wobj:=Wobj_Part_0;
		MoveL Tr_meulage_bavure_P98,[50,500,0,0],z0,Tool \wobj:=Wobj_Part_0;
		MoveL Tr_meulage_bavure_P99,[50,500,0,0],z0,Tool \wobj:=Wobj_Part_0;
		MoveL Tr_meulage_bavure_P100,[50,500,0,0],z0,Tool \wobj:=Wobj_Part_0;
		MoveL Tr_meulage_bavure_P101,[50,500,0,0],z0,Tool \wobj:=Wobj_Part_0;
		MoveL Tr_meulage_bavure_P102,[50,500,0,0],z0,Tool \wobj:=Wobj_Part_0;
		MoveL Tr_meulage_bavure_P103,[50,500,0,0],z0,Tool \wobj:=Wobj_Part_0;
		MoveL Tr_meulage_bavure_P104,[50,500,0,0],z0,Tool \wobj:=Wobj_Part_0;
		MoveL Tr_meulage_bavure_P105,[50,500,0,0],z0,Tool \wobj:=Wobj_Part_0;
		MoveL Tr_meulage_bavure_P106,[50,500,0,0],z0,Tool \wobj:=Wobj_Part_0;
		MoveL Tr_meulage_bavure_P107,[50,500,0,0],z0,Tool \wobj:=Wobj_Part_0;
		MoveL Tr_meulage_bavure_P108,[50,500,0,0],z0,Tool \wobj:=Wobj_Part_0;
		MoveL Tr_meulage_bavure_P109,[50,500,0,0],z0,Tool \wobj:=Wobj_Part_0;
		MoveL Tr_meulage_bavure_P110,[50,500,0,0],z0,Tool \wobj:=Wobj_Part_0;
		MoveL Tr_meulage_bavure_P111,[50,500,0,0],z0,Tool \wobj:=Wobj_Part_0;
		MoveL Tr_meulage_bavure_P112,[50,500,0,0],z0,Tool \wobj:=Wobj_Part_0;
		MoveL Tr_meulage_bavure_P113,[50,500,0,0],z0,Tool \wobj:=Wobj_Part_0;
		MoveL Tr_meulage_bavure_P114,[50,500,0,0],z0,Tool \wobj:=Wobj_Part_0;
		MoveL Tr_meulage_bavure_P115,[50,500,0,0],z0,Tool \wobj:=Wobj_Part_0;
		MoveL Tr_meulage_bavure_P116,[50,500,0,0],z0,Tool \wobj:=Wobj_Part_0;
		MoveL Tr_meulage_bavure_P117,[50,500,0,0],z0,Tool \wobj:=Wobj_Part_0;
		MoveL Tr_meulage_bavure_P118,[50,500,0,0],z0,Tool \wobj:=Wobj_Part_0;
		MoveL Tr_meulage_bavure_P119,[50,500,0,0],z0,Tool \wobj:=Wobj_Part_0;
		MoveL Tr_meulage_bavure_P120,[50,500,0,0],z0,Tool \wobj:=Wobj_Part_0;
		MoveL Tr_meulage_bavure_P121,[50,500,0,0],z0,Tool \wobj:=Wobj_Part_0;
		MoveL Tr_meulage_bavure_P122,[50,500,0,0],z0,Tool \wobj:=Wobj_Part_0;
		MoveL Tr_meulage_bavure_P123,[50,500,0,0],z0,Tool \wobj:=Wobj_Part_0;
		MoveL Tr_meulage_bavure_P124,[50,500,0,0],z0,Tool \wobj:=Wobj_Part_0;
		MoveL Tr_meulage_bavure_P125,[50,500,0,0],z0,Tool \wobj:=Wobj_Part_0;
		MoveL Tr_meulage_bavure_P126,[50,500,0,0],z0,Tool \wobj:=Wobj_Part_0;
		MoveL Tr_meulage_bavure_P127,[50,500,0,0],z0,Tool \wobj:=Wobj_Part_0;
		MoveL Tr_meulage_bavure_P128,[50,500,0,0],z0,Tool \wobj:=Wobj_Part_0;
		MoveL Tr_meulage_bavure_P129,[50,500,0,0],z0,Tool \wobj:=Wobj_Part_0;
		MoveL Tr_meulage_bavure_P130,[50,500,0,0],z0,Tool \wobj:=Wobj_Part_0;
		MoveL Tr_meulage_bavure_P131,[50,500,0,0],z0,Tool \wobj:=Wobj_Part_0;
		MoveL Tr_meulage_bavure_P132,[50,500,0,0],z0,Tool \wobj:=Wobj_Part_0;
		MoveL Tr_meulage_bavure_P133,[50,500,0,0],z0,Tool \wobj:=Wobj_Part_0;
		MoveL Tr_meulage_bavure_P134,[50,500,0,0],z0,Tool \wobj:=Wobj_Part_0;
		MoveL Tr_meulage_bavure_P135,[50,500,0,0],z0,Tool \wobj:=Wobj_Part_0;
		MoveL Tr_meulage_bavure_P136,[50,500,0,0],z0,Tool \wobj:=Wobj_Part_0;
		MoveL Tr_meulage_bavure_P137,[50,500,0,0],z0,Tool \wobj:=Wobj_Part_0;
		MoveL Tr_meulage_bavure_P138,[50,500,0,0],z0,Tool \wobj:=Wobj_Part_0;
		MoveL Tr_meulage_bavure_P139,[50,500,0,0],z0,Tool \wobj:=Wobj_Part_0;
		MoveL Tr_meulage_bavure_P140,[50,500,0,0],z0,Tool \wobj:=Wobj_Part_0;
		MoveL Tr_meulage_bavure_P141,[50,500,0,0],z0,Tool \wobj:=Wobj_Part_0;
		MoveL Tr_meulage_bavure_P142,[50,500,0,0],z0,Tool \wobj:=Wobj_Part_0;
		MoveL Tr_meulage_bavure_P143,[50,500,0,0],z0,Tool \wobj:=Wobj_Part_0;
		MoveL Tr_meulage_bavure_P144,[50,500,0,0],z0,Tool \wobj:=Wobj_Part_0;
		MoveL Tr_meulage_bavure_P145,[50,500,0,0],z0,Tool \wobj:=Wobj_Part_0;
		MoveL Tr_meulage_bavure_P146,[50,500,0,0],z0,Tool \wobj:=Wobj_Part_0;
		MoveL Tr_meulage_bavure_P147,[50,500,0,0],z0,Tool \wobj:=Wobj_Part_0;
		MoveL Tr_meulage_bavure_P148,[50,500,0,0],z0,Tool \wobj:=Wobj_Part_0;
		MoveL Tr_meulage_bavure_P149,[50,500,0,0],z0,Tool \wobj:=Wobj_Part_0;
		MoveL Tr_meulage_bavure_P150,[50,500,0,0],z0,Tool \wobj:=Wobj_Part_0;
		MoveL Tr_meulage_bavure_P151,[50,500,0,0],z0,Tool \wobj:=Wobj_Part_0;
		MoveL Tr_meulage_bavure_P152,[50,500,0,0],z0,Tool \wobj:=Wobj_Part_0;
		MoveL Tr_meulage_bavure_P153,[50,500,0,0],z0,Tool \wobj:=Wobj_Part_0;
		MoveL Tr_meulage_bavure_P154,[50,500,0,0],z0,Tool \wobj:=Wobj_Part_0;
		MoveL Tr_meulage_bavure_P155,[50,500,0,0],z0,Tool \wobj:=Wobj_Part_0;
		MoveL Tr_meulage_bavure_P156,[50,500,0,0],z0,Tool \wobj:=Wobj_Part_0;
		MoveL Tr_meulage_bavure_P157,[50,500,0,0],z0,Tool \wobj:=Wobj_Part_0;
		MoveL Tr_meulage_bavure_P158,[50,500,0,0],z0,Tool \wobj:=Wobj_Part_0;
		MoveL Tr_meulage_bavure_P159,[50,500,0,0],z0,Tool \wobj:=Wobj_Part_0;
		MoveL Tr_meulage_bavure_P160,[50,500,0,0],z0,Tool \wobj:=Wobj_Part_0;
		MoveL Tr_meulage_bavure_P161,[50,500,0,0],z0,Tool \wobj:=Wobj_Part_0;
		MoveL Tr_meulage_bavure_P162,[50,500,0,0],z0,Tool \wobj:=Wobj_Part_0;
		MoveL Tr_meulage_bavure_P163,[50,500,0,0],z0,Tool \wobj:=Wobj_Part_0;
		MoveL Tr_meulage_bavure_P164,[12.5,500,0,0],z0,Tool \wobj:=Wobj_Part_0;
		MoveL Tr_meulage_bavure_P165,[12.5,500,0,0],z0,Tool \wobj:=Wobj_Part_0;
		MoveL Tr_meulage_bavure_P166,[12.5,500,0,0],z0,Tool \wobj:=Wobj_Part_0;
		MoveL Tr_meulage_bavure_P167,[12.5,500,0,0],z0,Tool \wobj:=Wobj_Part_0;
		MoveL Tr_meulage_bavure_P168,[12.5,500,0,0],z0,Tool \wobj:=Wobj_Part_0;
		MoveL Tr_meulage_bavure_P169,[12.5,500,0,0],z0,Tool \wobj:=Wobj_Part_0;
		MoveL Tr_meulage_bavure_P170,[12.5,500,0,0],z0,Tool \wobj:=Wobj_Part_0;
		MoveL Tr_meulage_bavure_P171,[12.5,500,0,0],z0,Tool \wobj:=Wobj_Part_0;
		MoveL Tr_meulage_bavure_P172,[12.5,500,0,0],z0,Tool \wobj:=Wobj_Part_0;
		MoveL Tr_meulage_bavure_P173,[12.5,500,0,0],z0,Tool \wobj:=Wobj_Part_0;
		MoveL Tr_meulage_bavure_P174,[12.5,500,0,0],z0,Tool \wobj:=Wobj_Part_0;
		MoveL Tr_meulage_bavure_P175,[12.5,500,0,0],z0,Tool \wobj:=Wobj_Part_0;
		MoveL Tr_meulage_bavure_P176,[12.5,500,0,0],z0,Tool \wobj:=Wobj_Part_0;
		MoveL Tr_meulage_bavure_P177,[12.5,500,0,0],z0,Tool \wobj:=Wobj_Part_0;
		MoveL Tr_meulage_bavure_P178,[12.5,500,0,0],z0,Tool \wobj:=Wobj_Part_0;
		MoveL Tr_meulage_bavure_P179,[12.5,500,0,0],z0,Tool \wobj:=Wobj_Part_0;
		MoveL Tr_meulage_bavure_P180,[12.5,500,0,0],z0,Tool \wobj:=Wobj_Part_0;
		MoveL Tr_meulage_bavure_P181,[12.5,500,0,0],z0,Tool \wobj:=Wobj_Part_0;
		MoveL Tr_meulage_bavure_P182,[12.5,500,0,0],z0,Tool \wobj:=Wobj_Part_0;
		MoveL Tr_meulage_bavure_P183,[12.5,500,0,0],z0,Tool \wobj:=Wobj_Part_0;
		MoveL Tr_meulage_bavure_P184,[12.5,500,0,0],z0,Tool \wobj:=Wobj_Part_0;
		MoveL Tr_meulage_bavure_P185,[50,500,0,0],z0,Tool \wobj:=Wobj_Part_0;
		MoveL Tr_meulage_bavure_P186,[50,500,0,0],z0,Tool \wobj:=Wobj_Part_0;
		MoveL Tr_meulage_bavure_P187,[50,500,0,0],z0,Tool \wobj:=Wobj_Part_0;
		MoveL Tr_meulage_bavure_P188,[50,500,0,0],z0,Tool \wobj:=Wobj_Part_0;
		MoveL Tr_meulage_bavure_P189,[50,500,0,0],z0,Tool \wobj:=Wobj_Part_0;
		MoveL Tr_meulage_bavure_P190,[50,500,0,0],z0,Tool \wobj:=Wobj_Part_0;
		MoveL Tr_meulage_bavure_P191,[50,500,0,0],z0,Tool \wobj:=Wobj_Part_0;
		MoveL Tr_meulage_bavure_P192,[50,500,0,0],z0,Tool \wobj:=Wobj_Part_0;
		MoveL Tr_meulage_bavure_P193,[50,500,0,0],z0,Tool \wobj:=Wobj_Part_0;
		MoveL Tr_meulage_bavure_P194,[50,500,0,0],z0,Tool \wobj:=Wobj_Part_0;
		MoveL Tr_meulage_bavure_P195,[50,500,0,0],z0,Tool \wobj:=Wobj_Part_0;
		MoveL Tr_meulage_bavure_P196,[50,500,0,0],z0,Tool \wobj:=Wobj_Part_0;
		MoveL Tr_meulage_bavure_P197,[50,500,0,0],z0,Tool \wobj:=Wobj_Part_0;
		MoveL Tr_meulage_bavure_P198,[50,500,0,0],z0,Tool \wobj:=Wobj_Part_0;
		MoveL Tr_meulage_bavure_P199,[50,500,0,0],z0,Tool \wobj:=Wobj_Part_0;
		MoveL Tr_meulage_bavure_P200,[50,500,0,0],z0,Tool \wobj:=Wobj_Part_0;
		MoveL Tr_meulage_bavure_P201,[50,500,0,0],z0,Tool \wobj:=Wobj_Part_0;
		MoveL Tr_meulage_bavure_P202,[50,500,0,0],z0,Tool \wobj:=Wobj_Part_0;
		MoveL Tr_meulage_bavure_P203,[50,500,0,0],z0,Tool \wobj:=Wobj_Part_0;
		MoveL Tr_meulage_bavure_P204,[50,500,0,0],z0,Tool \wobj:=Wobj_Part_0;
		MoveL Tr_meulage_bavure_P205,[50,500,0,0],z0,Tool \wobj:=Wobj_Part_0;
		MoveL Tr_meulage_bavure_P206,[50,500,0,0],z0,Tool \wobj:=Wobj_Part_0;
		MoveL Tr_meulage_bavure_P207,[50,500,0,0],z0,Tool \wobj:=Wobj_Part_0;
		MoveL Tr_meulage_bavure_P208,[50,500,0,0],z0,Tool \wobj:=Wobj_Part_0;
		MoveL Tr_meulage_bavure_P209,[50,500,0,0],z0,Tool \wobj:=Wobj_Part_0;
		MoveL Tr_meulage_bavure_P210,[50,500,0,0],z0,Tool \wobj:=Wobj_Part_0;
		MoveL Tr_meulage_bavure_P211,[50,500,0,0],z0,Tool \wobj:=Wobj_Part_0;
		MoveL Tr_meulage_bavure_P212,[50,500,0,0],z0,Tool \wobj:=Wobj_Part_0;
		MoveL Tr_meulage_bavure_P213,[50,500,0,0],z0,Tool \wobj:=Wobj_Part_0;
		MoveL Tr_meulage_bavure_P214,[50,500,0,0],z0,Tool \wobj:=Wobj_Part_0;
		MoveL Tr_meulage_bavure_P215,[50,500,0,0],z0,Tool \wobj:=Wobj_Part_0;
		MoveL Tr_meulage_bavure_P216,[50,500,0,0],z0,Tool \wobj:=Wobj_Part_0;
		MoveL Tr_meulage_bavure_P217,[50,500,0,0],z0,Tool \wobj:=Wobj_Part_0;
		MoveL Tr_meulage_bavure_P218,[50,500,0,0],z0,Tool \wobj:=Wobj_Part_0;
		MoveL Tr_meulage_bavure_P219,[50,500,0,0],z0,Tool \wobj:=Wobj_Part_0;
		MoveL Tr_meulage_bavure_P220,[50,500,0,0],z0,Tool \wobj:=Wobj_Part_0;
		MoveL Tr_meulage_bavure_P221,[50,500,0,0],z0,Tool \wobj:=Wobj_Part_0;
		MoveL Tr_meulage_bavure_P222,[50,500,0,0],z0,Tool \wobj:=Wobj_Part_0;
		MoveL Tr_meulage_bavure_P223,[50,500,0,0],z0,Tool \wobj:=Wobj_Part_0;
		MoveL Tr_meulage_bavure_P224,[50,500,0,0],z0,Tool \wobj:=Wobj_Part_0;
		MoveL Tr_meulage_bavure_P225,[50,500,0,0],z0,Tool \wobj:=Wobj_Part_0;
		MoveL Tr_meulage_bavure_P226,[50,500,0,0],z0,Tool \wobj:=Wobj_Part_0;
		MoveL Tr_meulage_bavure_P227,[50,500,0,0],z0,Tool \wobj:=Wobj_Part_0;
		MoveL Tr_meulage_bavure_P228,[50,500,0,0],z0,Tool \wobj:=Wobj_Part_0;
		MoveL Tr_meulage_bavure_P229,[50,500,0,0],z0,Tool \wobj:=Wobj_Part_0;
		MoveL Tr_meulage_bavure_P230,[50,500,0,0],z0,Tool \wobj:=Wobj_Part_0;
		MoveL Tr_meulage_bavure_P231,[50,500,0,0],z0,Tool \wobj:=Wobj_Part_0;
		MoveL Tr_meulage_bavure_P232,[50,500,0,0],z0,Tool \wobj:=Wobj_Part_0;
		MoveL Tr_meulage_bavure_P233,[50,500,0,0],z0,Tool \wobj:=Wobj_Part_0;
		MoveL Tr_meulage_bavure_P234,[50,500,0,0],z0,Tool \wobj:=Wobj_Part_0;
		MoveL Tr_meulage_bavure_P235,[50,500,0,0],z0,Tool \wobj:=Wobj_Part_0;
		MoveL Tr_meulage_bavure_P236,[50,500,0,0],z0,Tool \wobj:=Wobj_Part_0;
		MoveL Tr_meulage_bavure_P237,[50,500,0,0],z0,Tool \wobj:=Wobj_Part_0;
		MoveL Tr_meulage_bavure_P238,[50,500,0,0],z0,Tool \wobj:=Wobj_Part_0;
		MoveL Tr_meulage_bavure_P239,[50,500,0,0],z0,Tool \wobj:=Wobj_Part_0;
		MoveL Tr_meulage_bavure_P240,[50,500,0,0],z0,Tool \wobj:=Wobj_Part_0;
		MoveL Tr_meulage_bavure_P241,[50,500,0,0],z0,Tool \wobj:=Wobj_Part_0;
		MoveL Tr_meulage_bavure_P242,[50,500,0,0],z0,Tool \wobj:=Wobj_Part_0;
		MoveL Tr_meulage_bavure_P243,[50,500,0,0],z0,Tool \wobj:=Wobj_Part_0;
		MoveL Tr_meulage_bavure_P244,[50,500,0,0],z0,Tool \wobj:=Wobj_Part_0;
		MoveL Tr_meulage_bavure_P245,[50,500,0,0],z0,Tool \wobj:=Wobj_Part_0;
		MoveL Tr_meulage_bavure_P246,[50,500,0,0],z0,Tool \wobj:=Wobj_Part_0;
		MoveL Tr_meulage_bavure_P247,[50,500,0,0],z0,Tool \wobj:=Wobj_Part_0;
		MoveL Tr_meulage_bavure_P248,[50,500,0,0],z0,Tool \wobj:=Wobj_Part_0;
		MoveL Tr_meulage_bavure_P249,[50,500,0,0],z0,Tool \wobj:=Wobj_Part_0;
		MoveL Tr_meulage_bavure_P250,[50,500,0,0],z0,Tool \wobj:=Wobj_Part_0;
		MoveL Tr_meulage_bavure_P251,[50,500,0,0],z0,Tool \wobj:=Wobj_Part_0;
		MoveL Tr_meulage_bavure_P252,[50,500,0,0],z0,Tool \wobj:=Wobj_Part_0;
		MoveL Tr_meulage_bavure_P253,[50,500,0,0],z0,Tool \wobj:=Wobj_Part_0;
		MoveL Tr_meulage_bavure_P254,[50,500,0,0],z0,Tool \wobj:=Wobj_Part_0;
		MoveL Tr_meulage_bavure_P255,[50,500,0,0],z0,Tool \wobj:=Wobj_Part_0;
		MoveL Tr_meulage_bavure_P256,[50,500,0,0],z0,Tool \wobj:=Wobj_Part_0;
		MoveL Tr_meulage_bavure_P257,[50,500,0,0],z0,Tool \wobj:=Wobj_Part_0;
		MoveL Tr_meulage_bavure_P258,[50,500,0,0],z0,Tool \wobj:=Wobj_Part_0;
		MoveL Tr_meulage_bavure_P259,[50,500,0,0],z0,Tool \wobj:=Wobj_Part_0;
		MoveL Tr_meulage_bavure_P260,[50,500,0,0],z0,Tool \wobj:=Wobj_Part_0;
		MoveL Tr_meulage_bavure_P261,[50,500,0,0],z0,Tool \wobj:=Wobj_Part_0;
		MoveL Tr_meulage_bavure_P262,[50,500,0,0],z0,Tool \wobj:=Wobj_Part_0;
		MoveL Tr_meulage_bavure_P263,[50,500,0,0],z0,Tool \wobj:=Wobj_Part_0;
		MoveL Tr_meulage_bavure_P264,[50,500,0,0],z0,Tool \wobj:=Wobj_Part_0;
		MoveL Tr_meulage_bavure_P265,[50,500,0,0],z0,Tool \wobj:=Wobj_Part_0;
		MoveL Tr_meulage_bavure_P266,[50,500,0,0],z0,Tool \wobj:=Wobj_Part_0;
		MoveL Tr_meulage_bavure_P267,[50,500,0,0],z0,Tool \wobj:=Wobj_Part_0;
		MoveL Tr_meulage_bavure_P268,[50,500,0,0],z0,Tool \wobj:=Wobj_Part_0;
		MoveL Tr_meulage_bavure_P269,[50,500,0,0],z0,Tool \wobj:=Wobj_Part_0;
		MoveL Tr_meulage_bavure_P270,[50,500,0,0],z0,Tool \wobj:=Wobj_Part_0;
		MoveL Tr_meulage_bavure_P271,[50,500,0,0],z0,Tool \wobj:=Wobj_Part_0;
		MoveL Tr_meulage_bavure_P272,[50,500,0,0],z0,Tool \wobj:=Wobj_Part_0;
		MoveL Tr_meulage_bavure_P273,[50,500,0,0],z0,Tool \wobj:=Wobj_Part_0;
		MoveL Tr_meulage_bavure_P274,[50,500,0,0],z0,Tool \wobj:=Wobj_Part_0;
		MoveL Tr_meulage_bavure_P275,[50,500,0,0],z0,Tool \wobj:=Wobj_Part_0;
		MoveL Tr_meulage_bavure_P276,[50,500,0,0],z0,Tool \wobj:=Wobj_Part_0;
		MoveL Tr_meulage_bavure_P277,[50,500,0,0],z0,Tool \wobj:=Wobj_Part_0;
		MoveL Tr_meulage_bavure_P278,[50,500,0,0],z0,Tool \wobj:=Wobj_Part_0;
		MoveL Tr_meulage_bavure_P279,[50,500,0,0],z0,Tool \wobj:=Wobj_Part_0;
		MoveL Tr_meulage_bavure_P280,[50,500,0,0],z0,Tool \wobj:=Wobj_Part_0;
		MoveL Tr_meulage_bavure_P281,[50,500,0,0],z0,Tool \wobj:=Wobj_Part_0;
		MoveL Tr_meulage_bavure_P282,[50,500,0,0],z0,Tool \wobj:=Wobj_Part_0;
		MoveL Tr_meulage_bavure_P283,[50,500,0,0],z0,Tool \wobj:=Wobj_Part_0;
		MoveL Tr_meulage_bavure_P284,[50,500,0,0],z0,Tool \wobj:=Wobj_Part_0;
		MoveL Tr_meulage_bavure_P285,[50,500,0,0],z0,Tool \wobj:=Wobj_Part_0;
		MoveL Tr_meulage_bavure_P286,[50,500,0,0],z0,Tool \wobj:=Wobj_Part_0;
		MoveL Tr_meulage_bavure_P287,[50,500,0,0],z0,Tool \wobj:=Wobj_Part_0;
		MoveL Tr_meulage_bavure_P288,[50,500,0,0],z0,Tool \wobj:=Wobj_Part_0;
		MoveL Tr_meulage_bavure_P289,[50,500,0,0],z0,Tool \wobj:=Wobj_Part_0;
		MoveL Tr_meulage_bavure_P290,[50,500,0,0],z0,Tool \wobj:=Wobj_Part_0;
		MoveL Tr_meulage_bavure_P291,[50,500,0,0],z0,Tool \wobj:=Wobj_Part_0;
		MoveL Tr_meulage_bavure_P292,[50,500,0,0],z0,Tool \wobj:=Wobj_Part_0;
		MoveL Tr_meulage_bavure_P293,[50,500,0,0],z0,Tool \wobj:=Wobj_Part_0;
		MoveL Tr_meulage_bavure_P294,[50,500,0,0],z0,Tool \wobj:=Wobj_Part_0;
		MoveJ Tr_meulage_bavure_degg1,V500,Z0,Tool,\Wobj:=Wobj_Part_0;
		MoveJ Tr_meulage_bavure_degg2,V2000,Z100,Tool,\Wobj:=Wobj_Part_0;
	ENDPROC
	 PROC P80_MAIN()
		Tr_pick;
		Tr_Cut;
		Tr_meulage_motif_1;
		Tr_meulage_bavure;
	ENDPROC
ENDMODULE
